FUNCTION_BLOCK FB_SetupArm
VAR_INPUT
END_VAR
VAR_OUTPUT
END_VAR
VAR
	// arm index, from 1 to 4
	m_armIdx: INT;
	
	// joints
	m_joints :ARRAY[1..g_sJntNum] OF FB_SetupJoint;
	
	// IO
	m_manualAdjustIO AT%I* :SINT;
	m_manualAdjustOnFlag :BOOL;
	m_autoAdjustIO AT%I* :SINT;
	m_autoAdjustDir :INT; // -1, 0, 1;
	
	// arm cartesian data, defined in cart origin
	m_curCartPose	:ST_Frame;
	
	// cartesion position of remote center
	m_rcPos :Vec3d;	
	
	// arm joint data
	m_curMotorPos :Vec5d;
	m_curLinkPos :Vec5d;
	m_curJntPos :Vec5d;
	m_curJntVel :Vec5d;
	m_curJntTrq :Vec5d;
	m_cmdJntTrq :Vec5d;
	m_rawJntCurrent :Vec5d;
	m_filtJntCurrent :Vec5d;
	m_cmdJntCurrent : Vec5d;
		
	// arm gravity
	m_jntGravity : Vec5d:=g_zeroVec5d;

	
END_VAR

PROPERTY armIdx : int
GET
armIdx:=m_armIdx;
END_GET
END_PROPERTY

// check auto adjust direction
METHOD autoAdjustDetect : INT
VAR_INPUT
END_VAR
// TODO
END_METHOD

PROPERTY autoAdjustDir : INT
GET
autoAdjustDir := m_autoAdjustDir;
END_GET
END_PROPERTY

METHOD checkIO : BOOL
VAR_INPUT
END_VAR
// check manual and auto adjust button
m_manualAdjustOnFlag := manualAdjustDetect();
m_autoAdjustDir :=autoAdjustDetect();
END_METHOD

PROPERTY cmdJntCurrent : REFERENCE TO  Vec5d
GET
cmdJntCurrent ref= m_cmdJntCurrent;
END_GET
END_PROPERTY

PROPERTY curCartPose : REFERENCE TO ST_Frame
GET
curCartPose ref=m_curCartPose;
END_GET
END_PROPERTY

PROPERTY curJntPos : REFERENCE TO Vec5d
GET
curJntPos ref=m_curJntPos;
END_GET
END_PROPERTY

PROPERTY curJntTrq : REFERENCE TO Vec5d
GET
curJntTrq ref=m_curJntTrq;
END_GET
END_PROPERTY

PROPERTY curJntVel :REFERENCE TO Vec5d
GET
curJntVel ref=m_curJntVel;
END_GET
END_PROPERTY

PROPERTY curLinkPos :REFERENCE TO Vec5d
GET
curLinkPos ref=m_curLinkPos;
END_GET
END_PROPERTY

PROPERTY curMotorPos : REFERENCE TO  Vec5d
GET
curMotorPos ref=m_curMotorPos;
END_GET
END_PROPERTY

METHOD PUBLIC enable : BOOL
VAR_IN_OUT CONSTANT
	i_jntIdx :Vec5i;
END_VAR
VAR
	i :INT ;
END_VAR
FOR i:=1 TO g_setupJntNum DO
	IF 1= i_jntIdx[i] THEN
		m_joints[i].enable();
	ELSE
		m_joints[i].disable();
	END_IF
END_FOR
END_METHOD

PROPERTY filtJntCurrent :REFERENCE TO Vec5d
GET
filtJntCurrent ref= m_filtJntCurrent;
END_GET
END_PROPERTY

// compute cartesion pose in cart origin
METHOD PROTECTED forwardKinematic : BOOL
VAR_IN_OUT CONSTANT
	i_jntPos :Vec5d;
END_VAR
VAR_IN_OUT
	r_cartPose :ST_Frame;
	
	// position of remote center
	r_rcPos :Vec3d;
END_VAR
VAR

END_VAR
//TODO
END_METHOD

METHOD PUBLIC init : BOOL
VAR_INPUT
	i_armIdx:INT;
END_VAR
VAR 
	i :INT ;
END_VAR
// arm statues init
m_armIdx:=i_armIdx;

// joint init
FOR i:=1 TO g_setupJntNum DO
	m_joints[i].init(m_armIdx, i);
END_FOR

// init joint encoder and position calculation
initJntPos();

// compute current status
updateStatus();
END_METHOD

METHOD initJntPos : BOOL
VAR_INPUT
END_VAR
VAR
	i:INT ;
END_VAR
// joint init
FOR i:=1 TO g_setupJntNum DO
	m_joints[i].initJntPos();
END_FOR
END_METHOD

// check if instrument is on
METHOD instruDetect : BOOL
VAR_INPUT
END_VAR
//TODO
END_METHOD

METHOD PUBLIC isEnabled : BOOL
VAR_IN_OUT CONSTANT
	i_jntIdx :Vec8i;
END_VAR
VAR
	i :INT ;
END_VAR
isEnabled := TRUE;
FOR i:=1 TO g_setupJntNum DO
	IF 1= i_jntIdx[i] THEN
		isEnabled :=  (m_joints[i].isEnabled() AND isEnabled);
	END_IF
END_FOR
END_METHOD

PROPERTY jntGravity :REFERENCE TO Vec5d
GET
jntGravity ref=m_jntGravity;
END_GET
END_PROPERTY

// check if adjust button is pressed
METHOD manualAdjustDetect : BOOL
VAR_INPUT
END_VAR
// TODO
END_METHOD

PROPERTY manualAdjustOn : bool
GET
manualAdjustOn := m_manualAdjustOnFlag;
END_GET
END_PROPERTY

PROPERTY rawJntCurrent :REFERENCE TO Vec5d
GET
rawJntCurrent ref=m_rawJntCurrent;
END_GET
END_PROPERTY

// update joints control command
METHOD PUBLIC updateCmds : BOOL
VAR_IN_OUT CONSTANT
	i_armCtrlCmd : ST_SetupArmCtrlCmds;
END_VAR
VAR
	i:INT;
END_VAR
m_cmdJntTrq:=i_armCtrlCmd.m_cmdJntTrq;

// enable/disable joints
enable(i_armCtrlCmd.m_jntEnableFlag);

// position/torque control
FOR i:=1 TO g_setupJntNum DO 
	IF i_armCtrlCmd.m_jntOPMode[i]=DriverOPMode_Trq THEN
		// gravity feedforward
		m_cmdJntTrq[i]:=m_cmdJntTrq[i]+m_jntGravity[i];
		m_joints[i].updateCmds(DriverOPMode_Trq,i_armCtrlCmd.m_cmdJntPos[i],m_cmdJntTrq[i]);
	ELSE
		m_cmdJntTrq[i]:=0;
		m_joints[i].updateCmds(DriverOPMode_Pos,i_armCtrlCmd.m_cmdJntPos[i],m_cmdJntTrq[i]);
	END_IF
	
END_FOR
END_METHOD

METHOD PUBLIC updateDyna : BOOL
VAR_IN_out constant
	i_jnt3Gravity :LREAL;
	i_jnt5Gravity :LREAL;
END_VAR
m_jntGravity[3]:=i_jnt3Gravity;
m_jntGravity[5]:=i_jnt5Gravity;
END_METHOD

// update arm status, including kinematic and dynamic
METHOD PUBLIC updateStatus : BOOL
VAR_INPUT
END_VAR
VAR 
	i,j:INT;
END_VAR
// update joint data
FOR i:=1 TO g_setupJntNum DO
	m_joints[i].updateStatus();
END_FOR

// check adjust button
checkIO();

// get joint data
FOR i:=1 TO g_setupJntNum DO
	m_curMotorPos[i]:=m_joints[i].motorPos;
	m_curLinkPos[i]:=m_joints[i].linkPos;
	m_curJntPos[i]:=m_joints[i].jntPos;
	m_curJntVel[i]:=m_joints[i].jntVel;
	m_curJntTrq[i]:=m_joints[i].jntTrq;
	m_rawJntCurrent[i]:=m_joints[i].rawCurrent;
	m_filtJntCurrent[i]:=m_joints[i].filtCurrent;
	m_cmdJntCurrent[i]:=m_joints[i].cmdCurrent;
END_FOR 

// cartesion pose
forwardKinematic(m_curJntPos,m_curCartPose,m_rcPos);
END_METHOD

END_FUNCTION_BLOCK

(* stored: Version 1.1.0.1, ProductVersion 3.1.4024.12
   POU FB_SetupArm: Id {5c9438f2-768b-4fff-9bfc-3693d995bd67}, SpecialFunc None
   Folder property: Id {c6ea0166-9703-475a-8e8e-3d0d51737a97}
   Property armIdx: Id {cabfa044-e4b7-4d76-b1b7-570e090205fc}
   Get Get: Id {5a987e19-0654-4dd3-bef9-5cc1d433e846}
   Method autoAdjustDetect: Id {c29550df-f892-45fc-bbea-033ea4e5f553}
   Property autoAdjustDir: Id {23463ad9-6b6b-4d71-8ec1-f29d801d18b3}
   Get Get: Id {11440852-0ab4-4acb-adbb-a37bb7e50412}
   Method checkIO: Id {fbd89c1b-d255-40db-a7aa-cd2a052b5167}
   Property cmdJntCurrent: Id {cf988543-58f5-435a-b7be-8f2740b3e7a6}
   Get Get: Id {00d8453b-1f45-4430-a6c7-bf4d2acc9ee1}
   Property curCartPose: Id {8b2d212c-f874-4df3-89c4-7a4c59a2497a}
   Get Get: Id {bff86ca2-da06-43d9-9418-b85d681657e9}
   Property curJntPos: Id {dce3bb79-9314-492e-9e98-fee04b74bd41}
   Get Get: Id {f8fadb86-6639-4fb2-a004-3b9df6fdd326}
   Property curJntTrq: Id {24ed19ef-7464-464e-880d-ef73a35a91a7}
   Get Get: Id {1774936a-ec78-4224-9f8a-11723c469020}
   Property curJntVel: Id {9c9eaed8-cbbc-4877-ac64-499b2f94549f}
   Get Get: Id {b341161a-d6a1-4f46-b87e-cd6dfc707fcd}
   Property curLinkPos: Id {31801798-9071-4878-9aba-12be0ad3e45d}
   Get Get: Id {246fe2c5-593e-4bd7-9156-a5d90d9026f6}
   Property curMotorPos: Id {2f4e185f-8286-482d-a2ae-9905a1d92411}
   Get Get: Id {970d1fb2-cdea-4a61-a53b-2160ac80684b}
   Method enable: Id {de5f38b7-8c95-4013-a120-bc96550e0d76}
   Property filtJntCurrent: Id {4315db90-bd10-4e4f-ab74-b8b2244311b8}
   Get Get: Id {9c348772-1b97-4208-9443-80c5fa591884}
   Method forwardKinematic: Id {49767c62-0ec4-4ada-b054-e0d81ad3f08d}
   Method init: Id {38d8d9c7-7db7-4b7f-9fc0-1defdd94f779}
   Method initJntPos: Id {2bf4e0ee-bb53-42fa-bd4c-c904be993a60}
   Method instruDetect: Id {58539efd-9cff-4819-9fe7-abe4f086c3a6}
   Method isEnabled: Id {b985692a-f6f7-460a-be8e-c41aacfdf6d5}
   Property jntGravity: Id {33c6cc0e-6d37-4855-b1be-0f076b081ccc}
   Get Get: Id {676c5d39-ab4d-45da-b342-fb30a86742c9}
   Method manualAdjustDetect: Id {9847d63f-214a-40a2-9f90-70dc67a85549}
   Property manualAdjustOn: Id {06fd6985-ca41-4e66-8b96-f30c8a6d0e2c}
   Get Get: Id {6b9e44f9-af7c-4368-b8c0-d50cceeb95b2}
   Property rawJntCurrent: Id {55d5ae20-b171-429a-ac31-06e15bf272af}
   Get Get: Id {6e301cc8-e411-4dac-b4d8-a08e42ea0f2d}
   Method updateCmds: Id {6d34fc6a-e3f4-42a7-8c5b-e82cddc386d1}
   Method updateDyna: Id {f00121ef-1617-4216-ab61-3a405eda46ec}
   Method updateStatus: Id {bb24dca5-7706-495a-abc4-658f70a32369} *)
